(* IEC 61131-3 sources: eCockpitGit/test_project/src/%F%00 Library/%F%Common Functions/%F%Math/%F%Percent Of, 1 file *)

(* ---- %POU%FU_iPerc_Of.st ---- *)
//This function calculates how many percent iA is of iOf
// +-----------+----------+----------+-----------------------------------------------------------------------------------------------------------------------+
// |**Version**|**Author**| **Date** |**Changes**                                                                                                            |
// +-----------+----------+----------+-----------------------------------------------------------------------------------------------------------------------+
// | 1         | NSN      | 08-09-17 | Creation                                                                                                              |
// +-----------+----------+----------+-----------------------------------------------------------------------------------------------------------------------+
// | 1.1       | NSN      | 20-11-17 | Added variable conversions to support e!Cockpit                                                                       |
// +-----------+----------+----------+-----------------------------------------------------------------------------------------------------------------------+
FUNCTION FU_iPerc_Of : INT
VAR_INPUT
	iA			:INT;		//The small value
	iOf			:INT;		//The big value
END_VAR
(*%!%__DELIMITER__%!%*)
FU_iPerc_Of			:=		TO_INT((TO_REAL(iA) / TO_REAL(iOf)) * 100);
